// TIA Portal V21 export
TYPE "Std_eTransferResponse"
   STRUCT
      reserved { ExternalVisible := 'False'} : Int;
      invalid_Channel { ExternalVisible := 'False'} : Int := 1;
      invlalid_TransferControl { ExternalVisible := 'False'} : Int := 2;
      invalid_AddressedTarget { ExternalVisible := 'False'} : Int := 3;
      invalid_Index { ExternalVisible := 'False'} : Int := 4;
      invalid_TransferValue { ExternalVisible := 'False'} : Int := 5;
      invalid_Combination { ExternalVisible := 'False'} : Int := 6;
      access_denied_DataInUse { ExternalVisible := 'False'} : Int := 7;
      no_data_empty_slot { ExternalVisible := 'False'} : Int := 8;
      invalid_ParameterSet { ExternalVisible := 'False'} : Int := 9;
      access_denied_WebConfig { ExternalVisible := 'False'} : Int := 10;
      access_denied_saving { ExternalVisible := 'False'} : Int := 11;
      no_valve_detected { ExternalVisible := 'False'} : Int := 15;
      reading_transfermode { ExternalVisible := 'False'} : Int := 20;
      ready_for_new_transfer { ExternalVisible := 'False'} : Int := 21;
      preparing_transfer { ExternalVisible := 'False'} : Int := 22;
      transferring { ExternalVisible := 'False'} : Int := 23;
      transfer_successful { ExternalVisible := 'False'} : Int := 24;
      FB_needs_rising_edge_xExecute { ExternalVisible := 'False'} : Int := 25;
      Valve_Mode_is_not_61_inactive { ExternalVisible := 'False'} : Int := 26;
      invalid_firmware_version { ExternalVisible := 'False'} : Int := 27;
      communication_failed { ExternalVisible := 'False'} : Int := 28;
      invalid_module_number { ExternalVisible := 'False'} : Int := 29;
      resetting { ExternalVisible := 'False'} : Int := 30;
      aborting { ExternalVisible := 'False'} : Int := 31;
   END_STRUCT;
END_TYPE
